SUBAPPLICATION mapping_aux (* Subapplication Type *)
  (* Standard: 61499-2 *)
  (* Version 1.0, 2023-01-29, Franz *)
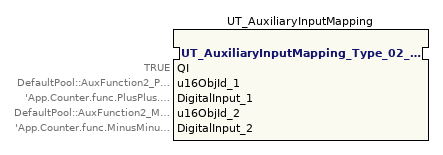
  FBS
    UT_AuxiliaryInputMapping : UT_AuxiliaryInputMapping_Type_02_Bool_NonLatched(QI := TRUE, u16ObjId_1 := DefaultPool::AuxFunction2_PlusPlus, DigitalInput_1 := 'App.Counter.func.PlusPlus.AuxFunction2', u16ObjId_2 := DefaultPool::AuxFunction2_MinusMinus, DigitalInput_2 := 'App.Counter.func.MinusMinus.AuxFunction2');
  END_FBS
END_SUBAPPLICATION
